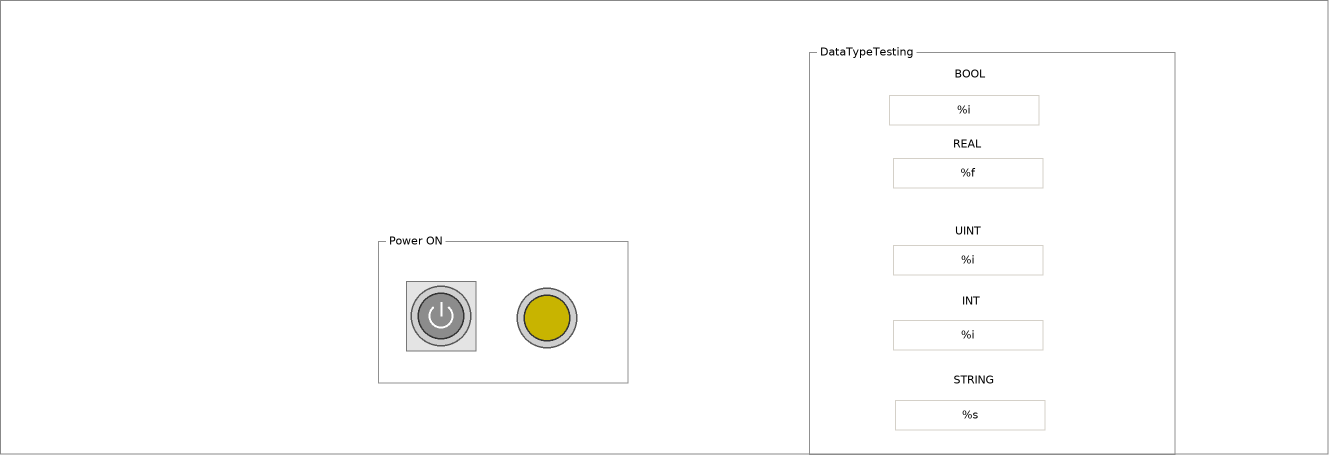
VISUALIZATION HMI  // 1329x455
    GroupBox (378,233 250x150), "Power ON"
        PowerSwitch (28,48 70x70), tooltip "Powerswitch", variable: MAIN.bStart, behaviour: TOGGLE, style: Switch-PowerSwitch-Gray
        Lamp1 (134,50 70x70), tooltip "light", variable: MAIN.bEnable, style: Lamp-Lamp1-Yellow
    GroupBox (809,44 366x411), "DataTypeTesting"
        Textfield (80,51 150x30), "%i", text variable: MAIN.nINT
        Textfield (84,114 150x30), "%f", text variable: MAIN.fREAL
        Textfield (84,276 150x30), "%i"
        Textfield (86,356 150x30), "%s"
        Textfield (84,201 150x30), "%i", text variable: MAIN.nUINT
        Label (86,15 150x30), "BOOL"
        Label (83,85 150x30), "REAL"
        Label (84,172 150x30), "UINT"
        Label (87,242 150x30), "INT"
        Label (90,321 150x30), "STRING"
    Label (1179,249 150x30)
END_VISUALIZATION

(* stored: Version 1.1.0.1, ProductVersion 3.1.4024.12
   Visu HMI: Id {cd5d7e0b-d33c-4fce-8df7-fffd92ded7fb} *)
